(* IEC 61131-3 sources: programs/VI-54/VI-54_20171205/VI-54_20171205/Stations/Screen/LseClass170718/Class/Logic_Or_10, 1 file *)

(* ---- Logic_Or_10.st ---- *)
(*!
<Class
	Name               = "Logic_Or_10"
	Revision           = "1.1"
	RealtimeTask       = "false"
	CyclicTask         = "false"
	BackgroundTask     = "false"
	Sigmatek           = "true"
	OSInterface        = "false"
	HighPriority       = "false"
	Automatic          = "false"
	UpdateMode         = "Prescan"
	IconPath           = ".\Class\Logic_Or_10\Logic_Or_Base.ico"
	SharedCommandTable = "true"
	Objectsize         = "(284,120)"
	Comment            = "V1.1 Logic OR class with 10 operands">
	<Channels>
		<Server
			Name           = "Result"
			Initialize     = "false"
			Visualized     = "true"
			WriteProtected = "true"
			Comment        = "If one client is &lt;&gt; 0 then result = 1">
		</Server>
		<Client Name="Op1" Required="false" Internal="false" Comment="Operand 1"/>
		<Client Name="Op10" Required="false" Internal="false" Comment="Operand 10"/>
		<Client Name="Op2" Required="false" Internal="false" Comment="Operand 2"/>
		<Client Name="Op3" Required="false" Internal="false" Comment="Operand 3"/>
		<Client Name="Op4" Required="false" Internal="false" Comment="Operand 4"/>
		<Client Name="Op5" Required="false" Internal="false" Comment="Operand 5"/>
		<Client Name="Op6" Required="false" Internal="false" Comment="Operand 6"/>
		<Client Name="Op7" Required="false" Internal="false" Comment="Operand 7"/>
		<Client Name="Op8" Required="false" Internal="false" Comment="Operand 8"/>
		<Client Name="Op9" Required="false" Internal="false" Comment="Operand 9"/>
	</Channels>
	<Network Name="Logic_Or_10">
		<!-- List of Components in this network -->
		<Components>
			<Object
				Name       = "_base"
				Class      = "Logic_Or_Base"
				Position   = "(810,1050)"
				Visualized = "true">
				<Channels>
					<Server Name="Result"/>
				</Channels>
			</Object>
		</Components>
		<Comments>
		</Comments>
		<!-- List of Connections in this network -->
		<Connections>
			<Connection Source="this.Result" Destination="_base.Result" Vertices="(1282,210),(1110,1140),"/>
		</Connections>
		<!-- Headerfiles -->
		<Options>
		</Options>
	</Network>
</Class>
*)
#pragma using Logic_Or_Base

Logic_Or_10 : CLASS
: Logic_Or_Base
  //Servers:
  //Clients:
	Op1 	: CltCh_DINT;
	Op2 	: CltCh_DINT;
	Op3 	: CltCh_DINT;
	Op4 	: CltCh_DINT;
	Op5 	: CltCh_DINT;
	Op6 	: CltCh_DINT;
	Op7 	: CltCh_DINT;
	Op8 	: CltCh_DINT;
	Op9 	: CltCh_DINT;
	Op10 	: CltCh_DINT;
  //Variables:
  //Functions:
  //Tables:
	FUNCTION @STD
		VAR_OUTPUT
			ret_code	: CONFSTATES;
		END_VAR;
	FUNCTION GLOBAL TAB @CT_;
END_CLASS;
